// TIA Portal V19 export
TYPE "OP_PB"
// stored: Access Published
   STRUCT
      Rest : Bool;
      Work : Bool;
   END_STRUCT;
END_TYPE
